(*==============================================================================================================================
CPNTeck - Automação industrial
(c)Copyright 2022 All Rights Reserved
_______________________________________________________________________________________________________________________________
Library: N/A 
Tested with: CX5140
Engineering: Twincat 3
Restrictions: -
Requirements: N/A
Functionality: This function block offers basic functionalities for distribute the positions generated from the program to the scoring toll
Support: fabio@cpnteck.com.br
Note: Parameter comments are only available in language 'English (United States)'
_______________________________________________________________________________________________________________________________
Change log table:

Version  		| Date        			| Expert in charge  	| Changes applied
01.00.01		| 29.03.2023  		| Fabio Campion            | First released version



===============================================================================================================================*)

(*Reset the scorer enabled array*)
FOR scorerEnabledIndex := 1 TO 20 BY 1 DO

	currentOrder.generatedOrder.scorerEnabledArr[scorerEnabledIndex] := FALSE;
	scorerPositionArr[scorerEnabledIndex] := 0;
	currentOrder.generatedOrder.scorerPositionReferenceArr[scorerEnabledIndex] := 0;

END_FOR;


scorerDistributionIndex := 1;
toolDistributionIndex := 2;
scorerExecTimes := 0;

(*Calculate the number of scorers to be used in the production*)

ACT_CalculateNumberOfScorers();


(*Distribute the scorer positions*)
IF currentOrder.generatedOrder.numberOfScorers > 0 THEN

	(*Distribute the scorer position for sheets with no scorer (Only count the sheets)*)
	IF currentOrder.order1.sheetType = SHEET_WITH_NO_SCORER THEN

		FOR scorerPositionTopIndex := 1 TO currentOrder.order1.sheetQuantity BY 1 DO

			toolDistributionIndex := toolDistributionIndex + 1;

		END_FOR

	END_IF

	(*Distribute the scorer position for sheets with two scorer*)
	IF currentOrder.order1.sheetType = SHEET_WITH_TWO_SCORER THEN

		scorerExecTimes := 0;

		FOR scorerPositionTopIndex := 1 TO currentOrder.order1.sheetQuantity BY 1 DO

			scorerExecTimes := scorerExecTimes + 1;

			scorerPositionArr[scorerDistributionIndex] := toolPositionArr[toolDistributionIndex];
			scorerDistributionIndex := scorerDistributionIndex + 1;
			toolDistributionIndex := toolDistributionIndex + 1;

			scorerPositionArr[scorerDistributionIndex] := toolPositionArr[toolDistributionIndex];
			scorerDistributionIndex := scorerDistributionIndex + 1;
			toolDistributionIndex := toolDistributionIndex + 2;

		END_FOR

	END_IF

	(*Distribute the scorer position for sheets with four scorer*)
	IF currentOrder.order1.sheetType = SHEET_WITH_FOUR_SCORER THEN

		scorerExecTimes :=0;

		FOR scorerPositionTopIndex := 1 TO currentOrder.order1.sheetQuantity BY 1 DO


			scorerPositionArr[scorerDistributionIndex] := toolPositionArr[toolDistributionIndex];
			scorerDistributionIndex := scorerDistributionIndex + 1;
			toolDistributionIndex := toolDistributionIndex + 1;

			scorerPositionArr[scorerDistributionIndex] := toolPositionArr[toolDistributionIndex];
			scorerDistributionIndex := scorerDistributionIndex + 1;
			toolDistributionIndex := toolDistributionIndex + 1;

			scorerPositionArr[scorerDistributionIndex] := toolPositionArr[toolDistributionIndex];
			scorerDistributionIndex := scorerDistributionIndex + 1;
			toolDistributionIndex := toolDistributionIndex + 1;

			scorerPositionArr[scorerDistributionIndex] := toolPositionArr[toolDistributionIndex];
			scorerDistributionIndex := scorerDistributionIndex + 1;
			toolDistributionIndex := toolDistributionIndex + 2;
			

		END_FOR

	END_IF

	(*Distribute the scorer position for sheets with two scorer - bottom orderr*)
	IF currentOrder.order2.sheetType = SHEET_WITH_TWO_SCORER THEN

		scorerExecTimes := 0;

		FOR scorerPositionBottomIndex := 1 TO currentOrder.order2.sheetQuantity BY 1 DO

			scorerExecTimes := scorerExecTimes + 1;

			scorerPositionArr[scorerDistributionIndex] := toolPositionArr[toolDistributionIndex];
			scorerDistributionIndex := scorerDistributionIndex + 1;
			toolDistributionIndex := toolDistributionIndex + 1;

			scorerPositionArr[scorerDistributionIndex] := toolPositionArr[toolDistributionIndex];
			scorerDistributionIndex := scorerDistributionIndex + 1;
			toolDistributionIndex := toolDistributionIndex + 2;

		END_FOR

	END_IF

	(*Distribute the scorer position for sheets with four scorer - bottom orderr*)
	IF currentOrder.order2.sheetType = SHEET_WITH_FOUR_SCORER THEN

		scorerExecTimes := 0;

		FOR scorerPositionBottomIndex := 1 TO currentOrder.order2.sheetQuantity BY 1 DO

			scorerPositionArr[scorerDistributionIndex] := toolPositionArr[toolDistributionIndex];
			scorerDistributionIndex := scorerDistributionIndex + 1;
			toolDistributionIndex := toolDistributionIndex + 1;

			scorerPositionArr[scorerDistributionIndex] := toolPositionArr[toolDistributionIndex];
			scorerDistributionIndex := scorerDistributionIndex + 1;
			toolDistributionIndex := toolDistributionIndex + 1;

			scorerPositionArr[scorerDistributionIndex] := toolPositionArr[toolDistributionIndex];
			scorerDistributionIndex := scorerDistributionIndex + 1;
			toolDistributionIndex := toolDistributionIndex + 1;

			scorerPositionArr[scorerDistributionIndex] := toolPositionArr[toolDistributionIndex];
			scorerDistributionIndex := scorerDistributionIndex + 1;
			toolDistributionIndex := toolDistributionIndex + 2;

		END_FOR

	END_IF

END_IF

//ACT_ScorerPositionDistribution();
_scorerPositionDistribution_1();
END_ACTION

END_FUNCTION_BLOCK

(* stored: Version 1.1.0.1
   POU FB_PositionsGeneration: Id {c9f902a4-8819-4eec-9e7b-f6614d83a996}, SpecialFunc None
   Method _bottomOrderDisplayControl: Id {2cf3d262-31e3-4555-8eb1-049ba0006094}
   Method _checkOrderLimits: Id {4093cb65-cbd9-4cec-9084-ac4019d348c7}
   Method _invertOrders: Id {fcc98153-3abc-4dd3-81c1-9bb682742fb9}
   Method _scorerPositionDistribution: Id {41254117-ebb4-474d-91e0-fca31a9e0b5a}
   Method _scorerPositionDistribution_1: Id {509f14ed-6470-4b3d-a6d1-9fa64dc318ed}
   Method _scorerPositionDistribution_bak: Id {e3bf6946-8eba-4a1c-904a-7a354f743995}
   Action ACT_CalculateNumberOfKnifes: Id {83872937-fac9-4e67-9872-1a4692ce9c10}
   Action ACT_CalculateNumberOfScorers: Id {80382a26-8d9d-407c-8175-e90058b01ef8}
   Action ACT_CalculateNumberOfSheets: Id {db769fe1-829e-4e71-add2-b7c58aa966e0}
   Action ACT_GenerateOrderPositions: Id {a149229c-bc8e-407c-8a99-84405415e883}
   Action ACT_KnifePositionDistribution: Id {b1fb4bc8-6d99-441a-bae5-102bc547fd35}
   Action ACT_KnifePositionDistribution_bak: Id {4b0cbfc6-c728-4f3d-832a-1dd1e9d6e22c}
   Action ACT_KnifePositionSelection: Id {0691d953-079b-454f-bf35-20fd03ccdc6c}
   Action ACT_ScorerPositionDistribution: Id {f682c022-9042-44a3-bec0-01ef0aa9a1db}
   Action ACT_ScorerPositionSelection: Id {14131191-f43e-4ad4-9138-b6130970c9a3} *)
